FUNCTION_BLOCK earth_fault (* Basic Function Block Type *)
  (* Standard: 61499-2 *)
  (* Version 0.0, 3/23/2016, gulzha, nxtControl GmbH, Template *)
  PACKAGE Main;
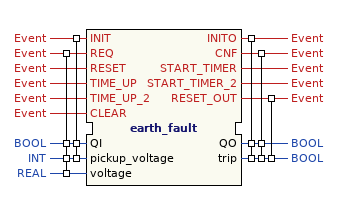
  EVENT_INPUT
    INIT WITH QI, pickup_voltage; (* Initialization Request *)
    REQ WITH QI, pickup_voltage, voltage; (* Normal Execution Request *)
    RESET;
    TIME_UP;
    TIME_UP_2;
    CLEAR;
  END_EVENT
  EVENT_OUTPUT
    INITO WITH QO, trip; (* Initialization Confirm *)
    CNF WITH QO, trip; (* Execution Confirmation *)
    START_TIMER;
    START_TIMER_2;
    RESET_OUT WITH trip;
  END_EVENT
  VAR_INPUT
    QI : BOOL; (* Input event qualifier *)
    pickup_voltage : INT;
    voltage : REAL;
  END_VAR
  VAR_OUTPUT
    QO : BOOL; (* Output event qualifier *)
    trip : BOOL;
  END_VAR
  VAR
    fault : BOOL;
  END_VAR
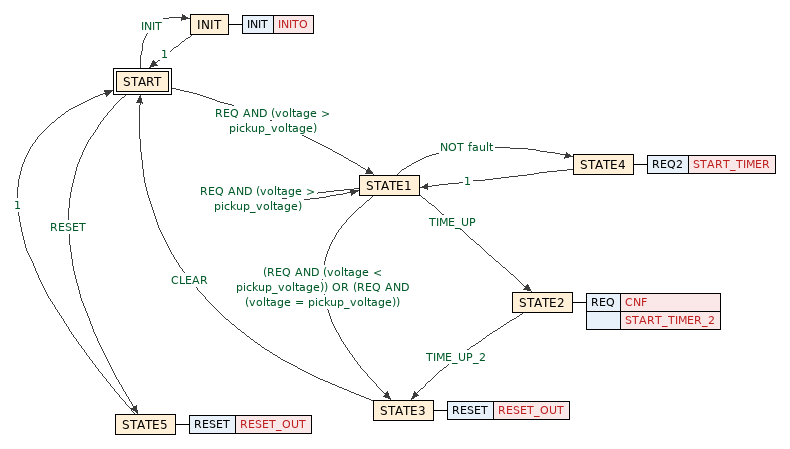
  EC_STATES
    START; (* Initial State *)
    INIT : INIT -> INITO; (* Initialization *)
    STATE1;
    STATE2 : REQ -> CNF, -> START_TIMER_2;
    STATE3 : RESET -> RESET_OUT;
    STATE4 : REQ2 -> START_TIMER;
    STATE5 : RESET -> RESET_OUT;
  END_STATES
  EC_TRANSITIONS
    START TO INIT := INIT;
    INIT TO START := 1;
    START TO STATE1 := REQ AND (voltage > pickup_voltage);
    STATE1 TO STATE2 := TIME_UP;
    STATE1 TO STATE3 := (REQ AND (voltage < pickup_voltage)) OR (REQ AND (voltage = pickup_voltage));
    STATE1 TO STATE1 := REQ AND (voltage > pickup_voltage);
    STATE2 TO STATE3 := TIME_UP_2;
    STATE5 TO START := 1;
    STATE1 TO STATE4 := NOT fault;
    STATE4 TO STATE1 := 1;
    START TO STATE5 := RESET;
    STATE3 TO START := CLEAR;
  END_TRANSITIONS
  ALGORITHM INIT IN ST: (* Initialization algorithm *)
;

trip := FALSE;
fault := FALSE;
  END_ALGORITHM
  ALGORITHM REQ IN ST: (* Normally executed algorithm *)
;
trip := TRUE;
  END_ALGORITHM
  ALGORITHM RESET IN ST:
;

trip := FALSE;
fault := FALSE;
  END_ALGORITHM
  ALGORITHM REQ2 IN ST:
;
fault := TRUE;
  END_ALGORITHM
END_FUNCTION_BLOCK
